(* LS Electric XG5000 project: test1 *)
(* PLC LSPLC *)
(* module base 0 slot 0: 입출력 모듈:XGH-DT4A (DC 24V 입력, 트랜지스터 출력 32점 ) *)

FUNCTION 시간검출 : ARRAY[0..5] OF WORD
VAR_INPUT
    _RTC_TIME_0 : BYTE;
    _RTC_TIME_1 : BYTE;
    _RTC_TIME_2 : BYTE;
    _RTC_TIME_3 : BYTE;
    _RTC_TIME_4 : BYTE;
    _RTC_TIME_5 : BYTE;
END_VAR

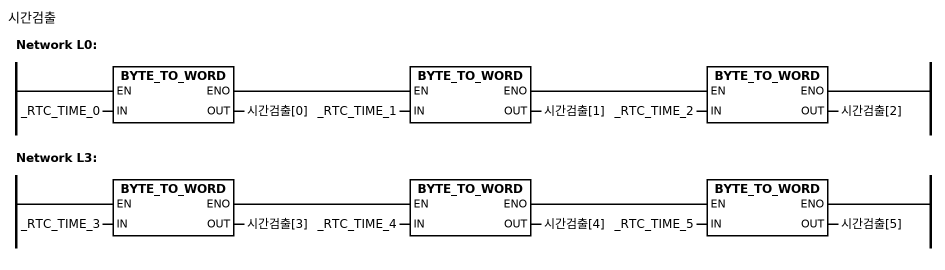
(* Rung L0 *)
시간검출[0] := BYTE_TO_WORD(_RTC_TIME_0);
시간검출[1] := BYTE_TO_WORD(_RTC_TIME_1);
시간검출[2] := BYTE_TO_WORD(_RTC_TIME_2);
(* Rung L3 *)
시간검출[3] := BYTE_TO_WORD(_RTC_TIME_3);
시간검출[4] := BYTE_TO_WORD(_RTC_TIME_4);
시간검출[5] := BYTE_TO_WORD(_RTC_TIME_5);
END_FUNCTION

PROGRAM NewProgram (* task: 스캔 프로그램 *)
VAR
    in1 : BOOL;
    in2 : WORD;
    in3 : BOOL;
    in4 : BOOL;
    in5 : BOOL;
    in6 : BOOL;
    in7 : BOOL;
    in8 : BOOL;
    in9 : BOOL;
    INST : TON;
    move_i : INT;
    move_in : BOOL;
    move_o : INT;
    move_out : BOOL;
    out1 : BOOL;
    out2 : BOOL;
    out3 : BOOL;
    out4 : BOOL;
    out5 : BOOL;
    out6 : BOOL;
    t1 : TON;
    t1_out : BOOL;
    t1_switch : BOOL;
    t2 : TON;
    t3 : TON;
    t3_램프 : BOOL;
    t4 : TON;
    time1 : TIME;
    time1_out : TIME;
    time_out : WORD;
    ton_in : BOOL;
    ton_out : BOOL;
    trigger : BOOL;
    결과1 : INT;
    결과1_R : REAL;
    년 : WORD;
    램프 : BOOL;
    물 : BOOL;
    물1 : BOOL;
    물2 : BOOL;
    변기 : BOOL;
    센서 : BOOL;
    숫자1 : INT;
    숫자1_R : REAL;
    스위치 : BOOL;
    시간검출 : ARRAY[0..5] OF WORD;
    시간검출_out : WORD;
    실습1_switch : BOOL;
    실습1_t1 : TON;
    실습1_t2 : TOF;
    실습1_램프 : BOOL;
    실습2_switch : BOOL;
    실습2_t1 : TON;
    실습2_t1_switch : BOOL;
    실습2_t2 : TON;
    실습2_t2_switch : BOOL;
    실습2_t3 : TON;
    실습2_t3_switch : BOOL;
    실습2_t3_램프 : BOOL;
    실습2_t4_switch : BOOL;
    실습2_tp1 : TP;
    실습2_tp2 : TP;
    실습2_tp3 : TP;
    실습2_tp4 : TP;
    월 : WORD;
    일 : WORD;
    입력 : BOOL;
END_VAR
VAR
    _e1 : R_TRIG;
    _e2 : R_TRIG;
    _e3 : R_TRIG;
END_VAR

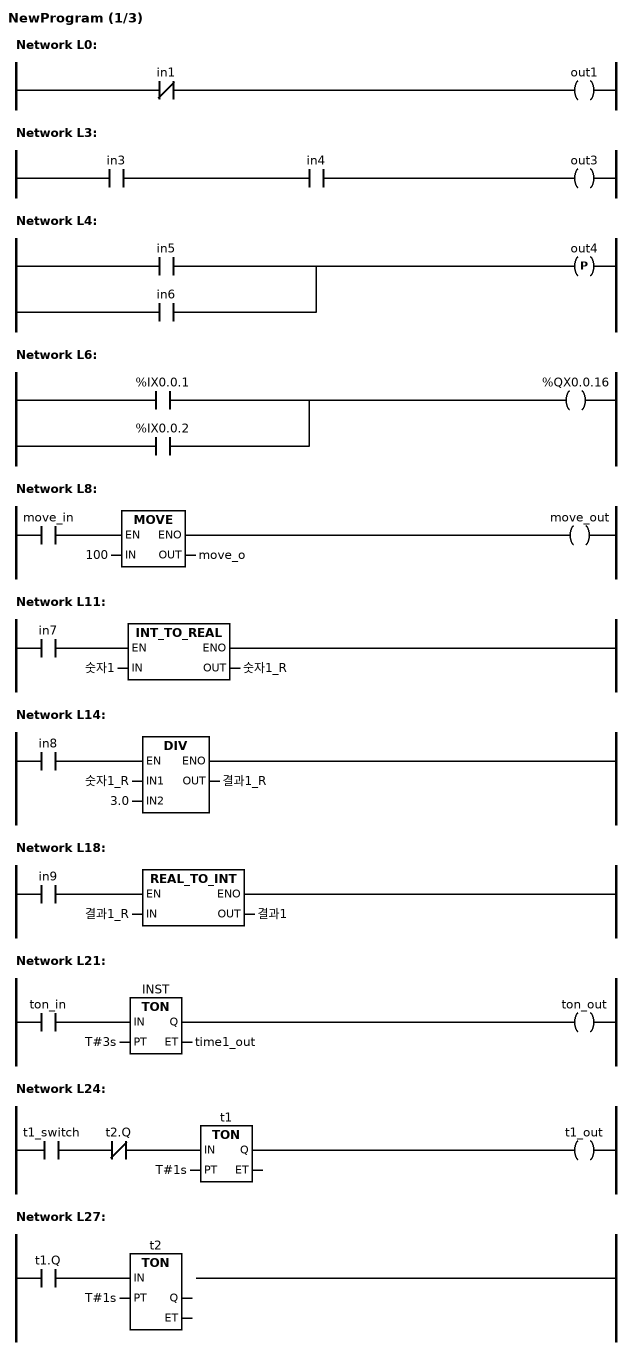
(* Rung L0 *)
out1 := NOT in1;
(* Rung L3 *)
out3 := in3 AND in4;
(* Rung L4 *)
_e1(CLK := in5 OR in6);
out4 := _e1.Q;
(* Rung L6 *)
%QX0.0.16 := %IX0.0.1 OR %IX0.0.2;
(* Rung L8 *)
IF move_in THEN move_o := 100; END_IF;
move_out := move_in;
(* Rung L11 *)
IF in7 THEN 숫자1_R := INT_TO_REAL(숫자1); END_IF;
(* Rung L14 *)
IF in8 THEN 결과1_R := 숫자1_R / 3.0; END_IF;
(* Rung L18 *)
IF in9 THEN 결과1 := REAL_TO_INT(결과1_R); END_IF;
(* Rung L21 *)
INST(IN := ton_in, PT := T#3s, ET => time1_out);
ton_out := INST.Q;
(* Rung L24 *)
t1(IN := t1_switch AND NOT t2.Q, PT := T#1s);
t1_out := t1.Q;
(* Rung L27 *)
t2(IN := t1.Q, PT := T#1s);

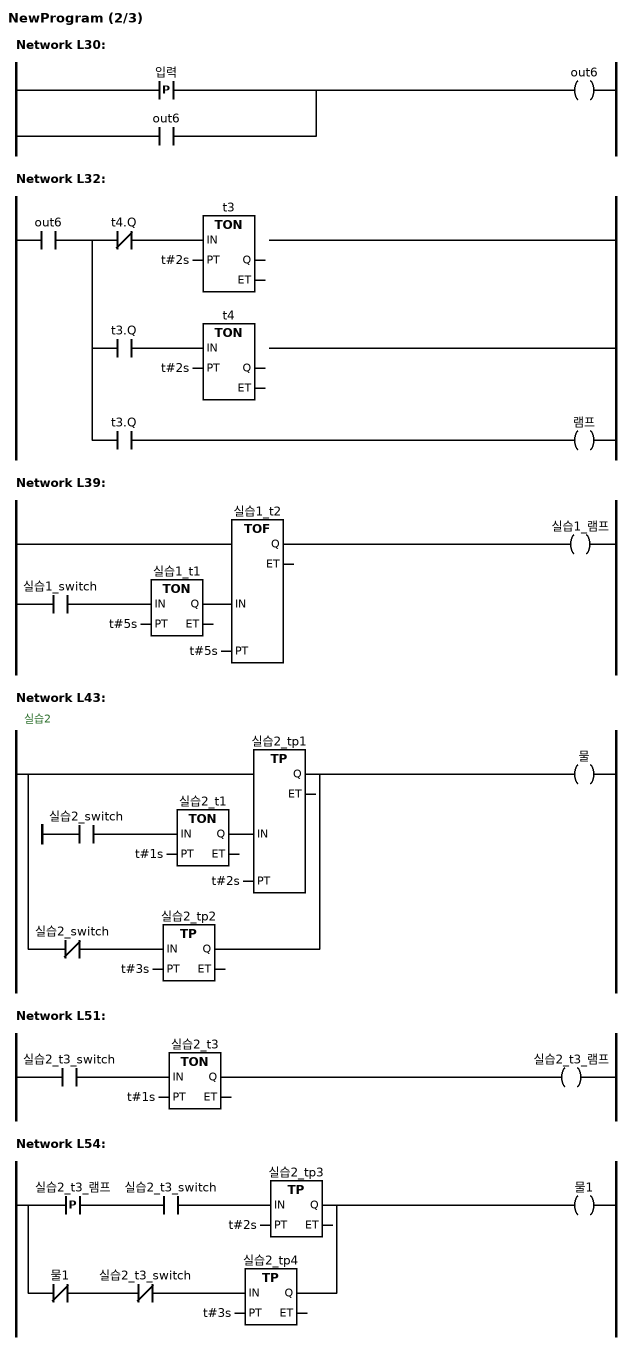
(* Rung L30 *)
_e2(CLK := 입력);
out6 := _e2.Q OR out6;
(* Rung L32 *)
t3(IN := out6 AND NOT t4.Q, PT := t#2s);
t4(IN := out6 AND t3.Q, PT := t#2s);
램프 := out6 AND t3.Q;
(* Rung L39 *)
실습1_t1(IN := 실습1_switch, PT := t#5s);
실습1_t2(IN := 실습1_t1.Q, PT := t#5s);
실습1_램프 := 실습1_t2.Q;
(* 실습2 *)
(* Rung L43 *)
실습2_t1(IN := 실습2_switch, PT := t#1s);
실습2_tp1(IN := 실습2_t1.Q, PT := t#2s);
실습2_tp2(IN := NOT 실습2_switch, PT := t#3s);
물 := 실습2_tp1.Q OR 실습2_tp2.Q;
(* Rung L51 *)
실습2_t3(IN := 실습2_t3_switch, PT := t#1s);
실습2_t3_램프 := 실습2_t3.Q;
(* Rung L54 *)
_e3(CLK := 실습2_t3_램프);
실습2_tp3(IN := _e3.Q AND 실습2_t3_switch, PT := t#2s);
실습2_tp4(IN := NOT 물1 AND NOT 실습2_t3_switch, PT := t#3s);
물1 := 실습2_tp3.Q OR 실습2_tp4.Q;

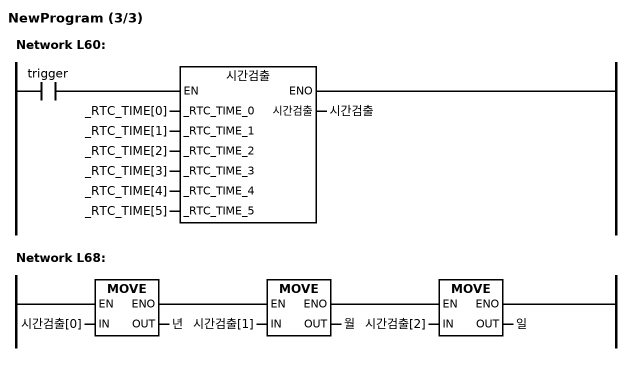
(* Rung L60 *)
IF trigger THEN
    시간검출 := 시간검출(_RTC_TIME_0 := _RTC_TIME[0], _RTC_TIME_1 := _RTC_TIME[1], _RTC_TIME_2 := _RTC_TIME[2], _RTC_TIME_3 := _RTC_TIME[3], _RTC_TIME_4 := _RTC_TIME[4], _RTC_TIME_5 := _RTC_TIME[5]);
END_IF;
(* Rung L68 *)
년 := 시간검출[0];
월 := 시간검출[1];
일 := 시간검출[2];
END_PROGRAM